Staubli VAL3: OnF5.pgx

public program OnF5()
begin
end
